PROGRAM MAIN
VAR
	iCurrentTemp : INT;
	iSetTemp : INT;
	bheating AT %Q*: BOOL := FALSE;
	iInputsettemp AT %I*: INT;
	iInputcurrenttemp AT %I*: INT;
	
	fb1HZ: TON := (PT := TIME#1S0MS);
	TemperatureTable: ARRAY[1..20] OF INT := [0, 0, 0, 0, 0, 0, 0, 0, 0, 0, 0, 0, 0, 0, 0, 0, 0, 0, 0, 0];
	Index: INT := 1;
	sr: TON;
END_VAR

iSetTemp :=  LREAL_TO_INT(F_Scale(iInputsettemp,0,32767,10,30));
iCurrentTemp :=  LREAL_TO_INT(F_Scale(iInputcurrenttemp,0,32767,-30,40));
fb1HZ(IN:= NOT(fb1HZ.Q));
IF fb1HZ.Q THEN
	TemperatureTable[Index] := iCurrentTemp;
	Index := Index +1;
	IF index = 21 THEN
		index := 1;
	END_IF
END_IF
IF iSetTemp > iCurrentTemp  THEN
	bheating := TRUE;
ELSE
	bheating := FALSE;
END_IF

END_PROGRAM

(* stored: Version 1.1.0.1, ProductVersion 3.1.4024.12
   POU MAIN: Id {2d2c30b1-4b8e-40fd-b0de-3d5b86e5415d}, SpecialFunc None *)
